// TIA Portal V18 export
FUNCTION_BLOCK "FB1-MR_Flowrate Control"   // FB1, LAD
{ S7_Optimized_Access := 'TRUE' }
VERSION : 0.1
// stored: AutoNumber true, IsIECCheckEnabled false, IsRetainMemResEnabled false, MemoryReserve 100, SetENOAutomatically false, UDAEnableTagReadback false
   VAR_INPUT
      "Pump size A" : Real;
      "pump size B" : Real;
      "Pump speed A" : Real;
      "pump Speed B" : Real;
      "Mixing Ratio 100:B" : Real;
      "Metering Qty" : Real;
      "Metering Flowrate" : Real;
      "Flowrate Adjustemnt A %" : Real;
      "Flowrate Adjustment B %" : Real;
      "Pump A max Hz" : Real;
      "pump B max Hz" : Real;
   END_VAR
   VAR_OUTPUT
      "Flowrate pump A without adjustment" : Real;
      "Flowrate pump B without adjustment" : Real;
      "Flowrate pump A with adjustment" : Real;
      "Flowrate pump B with adjustment" : Real;
      "Mixed Flowrate" : Real;
      "Pump Capacity A cc/min" : Real;
      "Pump capacity B cc/min" : Real;
      "Pump A frequency" : Real;
      "Pump B frequency" : Real;
      "Metering time" : DInt;
      "Meteringtime in sec" : Int;
   END_VAR
   VAR
      "Maximum Flowrate Pump A" : Real;
      "Maximum Flowrate Pump B" : Real;
      "Pump compensation" : Real;
      "Individual flowrate A MR" : Real;
      "Individual flowrate B1 MR" : Real;
      "Individual flowrate B MR" : Real;
      "Flowrate Ratio difference A" : Real;
      "Flowrate Ratio difference B" : Real;
      "Flowrate Pump A" : Real;
      "Flowrate Pump B" : Real;
      "Flowrate B After Compensation" : Real;
      "Mixed flowrate A+B" : Real;
      "Flowrate to adjust A" : Real;
      "Flowrate to adjust B" : Real;
      "metering time in minutes" : Real;
      "metering time in Sec" : Real;
      "Metering time in msec" : LReal;
      "flowrate to adjust A_1" : Real;
      "flowrate to adjust B_1" : Real;
      "Ratio>100" : Real;
      "amount to reduce in A" : Real;
      "Flowrate difference" : Real;
      "Ratio margin" : Real;
      "Ratio/100" : Real;
      "Flowrate A Per ratio" : Real;
      "A Flowrate Compensated" : Real;
   END_VAR
BEGIN

REGION Network 1: Pump Size and speed multiplication
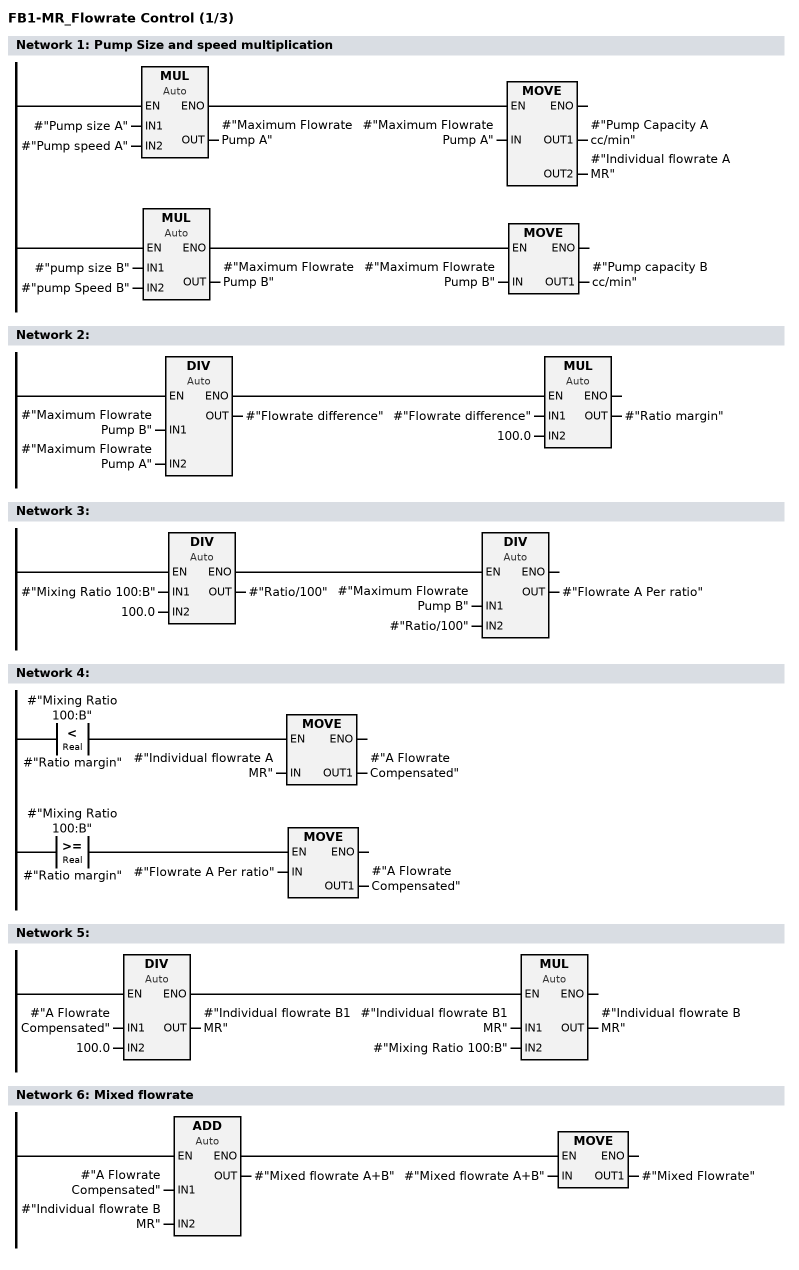
   RUNG wire#powerrail
      Mul(in1 := #"Pump size A", in2 := #"Pump speed A", out => #"Maximum Flowrate Pump A")
      Move(in := #"Maximum Flowrate Pump A", out1 => #"Pump Capacity A cc/min", out2 => #"Individual flowrate A MR")
   END_RUNG
   RUNG wire#powerrail
      Mul(in1 := #"pump size B", in2 := #"pump Speed B", out => #"Maximum Flowrate Pump B")
      Move(in := #"Maximum Flowrate Pump B", out1 => #"Pump capacity B cc/min")
   END_RUNG
   // the same network as SCL:
   #"Maximum Flowrate Pump A" := #"Pump size A" * #"Pump speed A";
   #"Pump Capacity A cc/min" := #"Maximum Flowrate Pump A";
   #"Individual flowrate A MR" := #"Maximum Flowrate Pump A";
   #"Maximum Flowrate Pump B" := #"pump size B" * #"pump Speed B";
   #"Pump capacity B cc/min" := #"Maximum Flowrate Pump B";
END_REGION

REGION Network 2
   RUNG wire#powerrail
      Div(in1 := #"Maximum Flowrate Pump B", in2 := #"Maximum Flowrate Pump A", out => #"Flowrate difference")
      Mul(in1 := #"Flowrate difference", in2 := 100.0, out => #"Ratio margin")
   END_RUNG
   // the same network as SCL:
   #"Flowrate difference" := #"Maximum Flowrate Pump B" / #"Maximum Flowrate Pump A";
   #"Ratio margin" := #"Flowrate difference" * 100.0;
END_REGION

REGION Network 3
   RUNG wire#powerrail
      Div(in1 := #"Mixing Ratio 100:B", in2 := 100.0, out => #"Ratio/100")
      Div(in1 := #"Maximum Flowrate Pump B", in2 := #"Ratio/100", out => #"Flowrate A Per ratio")
   END_RUNG
   // the same network as SCL:
   #"Ratio/100" := #"Mixing Ratio 100:B" / 100.0;
   #"Flowrate A Per ratio" := #"Maximum Flowrate Pump B" / #"Ratio/100";
END_REGION

REGION Network 4
   RUNG wire#powerrail
      { S7_Templates := "SrcType := Real" } LT_Contact(in1 := #"Mixing Ratio 100:B", in2 := #"Ratio margin")
      Move(in := #"Individual flowrate A MR", out1 => #"A Flowrate Compensated")
   END_RUNG
   RUNG wire#powerrail
      { S7_Templates := "SrcType := Real" } GE_Contact(in1 := #"Mixing Ratio 100:B", in2 := #"Ratio margin")
      Move(in := #"Flowrate A Per ratio", out1 => #"A Flowrate Compensated")
   END_RUNG
   // the same network as SCL:
   IF #"Mixing Ratio 100:B" < #"Ratio margin" THEN
       #"A Flowrate Compensated" := #"Individual flowrate A MR";
   END_IF;
   IF #"Mixing Ratio 100:B" >= #"Ratio margin" THEN
       #"A Flowrate Compensated" := #"Flowrate A Per ratio";
   END_IF;
END_REGION

REGION Network 5
   RUNG wire#powerrail
      Div(in1 := #"A Flowrate Compensated", in2 := 100.0, out => #"Individual flowrate B1 MR")
      Mul(in1 := #"Individual flowrate B1 MR", in2 := #"Mixing Ratio 100:B", out => #"Individual flowrate B MR")
   END_RUNG
   // the same network as SCL:
   #"Individual flowrate B1 MR" := #"A Flowrate Compensated" / 100.0;
   #"Individual flowrate B MR" := #"Individual flowrate B1 MR" * #"Mixing Ratio 100:B";
END_REGION

REGION Network 6: Mixed flowrate
   RUNG wire#powerrail
      Add(in1 := #"A Flowrate Compensated", in2 := #"Individual flowrate B MR", out => #"Mixed flowrate A+B")
      Move(in := #"Mixed flowrate A+B", out1 => #"Mixed Flowrate")
   END_RUNG
   // the same network as SCL:
   #"Mixed flowrate A+B" := #"A Flowrate Compensated" + #"Individual flowrate B MR";
   #"Mixed Flowrate" := #"Mixed flowrate A+B";
END_REGION

REGION Network 7: flowrate ratio difference
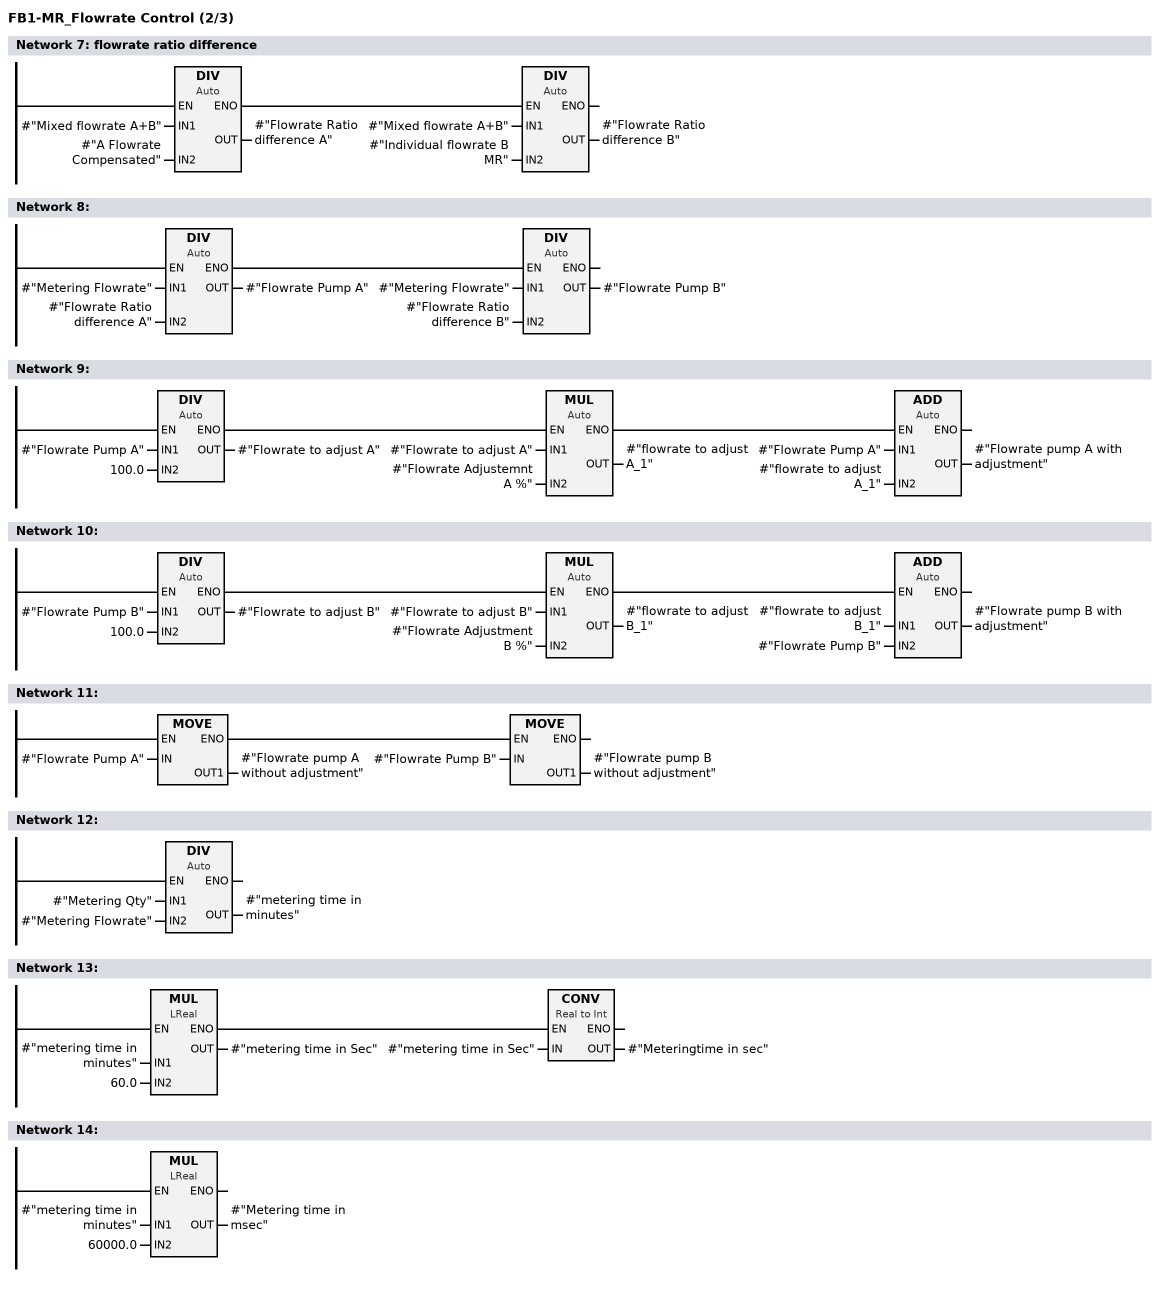
   RUNG wire#powerrail
      Div(in1 := #"Mixed flowrate A+B", in2 := #"A Flowrate Compensated", out => #"Flowrate Ratio difference A")
      Div(in1 := #"Mixed flowrate A+B", in2 := #"Individual flowrate B MR", out => #"Flowrate Ratio difference B")
   END_RUNG
   // the same network as SCL:
   #"Flowrate Ratio difference A" := #"Mixed flowrate A+B" / #"A Flowrate Compensated";
   #"Flowrate Ratio difference B" := #"Mixed flowrate A+B" / #"Individual flowrate B MR";
END_REGION

REGION Network 8
   RUNG wire#powerrail
      Div(in1 := #"Metering Flowrate", in2 := #"Flowrate Ratio difference A", out => #"Flowrate Pump A")
      Div(in1 := #"Metering Flowrate", in2 := #"Flowrate Ratio difference B", out => #"Flowrate Pump B")
   END_RUNG
   // the same network as SCL:
   #"Flowrate Pump A" := #"Metering Flowrate" / #"Flowrate Ratio difference A";
   #"Flowrate Pump B" := #"Metering Flowrate" / #"Flowrate Ratio difference B";
END_REGION

REGION Network 9
   RUNG wire#powerrail
      Div(in1 := #"Flowrate Pump A", in2 := 100.0, out => #"Flowrate to adjust A")
      Mul(in1 := #"Flowrate to adjust A", in2 := #"Flowrate Adjustemnt A %", out => #"flowrate to adjust A_1")
      Add(in1 := #"Flowrate Pump A", in2 := #"flowrate to adjust A_1", out => #"Flowrate pump A with adjustment")
   END_RUNG
   // the same network as SCL:
   #"Flowrate to adjust A" := #"Flowrate Pump A" / 100.0;
   #"flowrate to adjust A_1" := #"Flowrate to adjust A" * #"Flowrate Adjustemnt A %";
   #"Flowrate pump A with adjustment" := #"Flowrate Pump A" + #"flowrate to adjust A_1";
END_REGION

REGION Network 10
   RUNG wire#powerrail
      Div(in1 := #"Flowrate Pump B", in2 := 100.0, out => #"Flowrate to adjust B")
      Mul(in1 := #"Flowrate to adjust B", in2 := #"Flowrate Adjustment B %", out => #"flowrate to adjust B_1")
      Add(in1 := #"flowrate to adjust B_1", in2 := #"Flowrate Pump B", out => #"Flowrate pump B with adjustment")
   END_RUNG
   // the same network as SCL:
   #"Flowrate to adjust B" := #"Flowrate Pump B" / 100.0;
   #"flowrate to adjust B_1" := #"Flowrate to adjust B" * #"Flowrate Adjustment B %";
   #"Flowrate pump B with adjustment" := #"flowrate to adjust B_1" + #"Flowrate Pump B";
END_REGION

REGION Network 11
   RUNG wire#powerrail
      Move(in := #"Flowrate Pump A", out1 => #"Flowrate pump A without adjustment")
      Move(in := #"Flowrate Pump B", out1 => #"Flowrate pump B without adjustment")
   END_RUNG
   // the same network as SCL:
   #"Flowrate pump A without adjustment" := #"Flowrate Pump A";
   #"Flowrate pump B without adjustment" := #"Flowrate Pump B";
END_REGION

REGION Network 12
   RUNG wire#powerrail
      Div(in1 := #"Metering Qty", in2 := #"Metering Flowrate", out => #"metering time in minutes")
   END_RUNG
   // the same network as SCL:
   #"metering time in minutes" := #"Metering Qty" / #"Metering Flowrate";
END_REGION

REGION Network 13
   RUNG wire#powerrail
      { S7_Templates := "SrcType := LReal" } Mul(in1 := #"metering time in minutes", in2 := 60.0, out => #"metering time in Sec")
      { S7_Templates := "[SrcType := Real, DestType := Int]" } Convert(in := #"metering time in Sec", out => #"Meteringtime in sec")
   END_RUNG
   // the same network as SCL:
   #"metering time in Sec" := #"metering time in minutes" * 60.0;
   #"Meteringtime in sec" := REAL_TO_INT(#"metering time in Sec");
END_REGION

REGION Network 14
   RUNG wire#powerrail
      { S7_Templates := "SrcType := LReal" } Mul(in1 := #"metering time in minutes", in2 := 60000.0, out => #"Metering time in msec")
   END_RUNG
   // the same network as SCL:
   #"Metering time in msec" := #"metering time in minutes" * 60000.0;
END_REGION

REGION Network 15
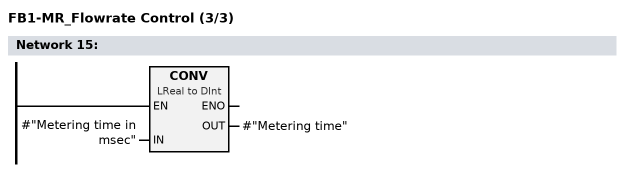
   RUNG wire#powerrail
      { S7_Templates := "[SrcType := LReal, DestType := DInt]" } Convert(in := #"Metering time in msec", out => #"Metering time")
   END_RUNG
   // the same network as SCL:
   #"Metering time" := LREAL_TO_DINT(#"Metering time in msec");
END_REGION
END_FUNCTION_BLOCK
